VAR_GLOBAL CONSTANT
	cuinMaxConnections: UINT := 50;
END_VAR

(* stored: Version 1.1.0.1, ProductVersion 3.1.4019.2
   GVL ACL_Const: Id {c8d6b96f-e5c4-4b10-b8bc-2f87add6d659} *)
